KUKA KRL program: ps_p13060r5_ltc_geo_c1.src, ps_p13060r5_ltc_geo_c1.dat

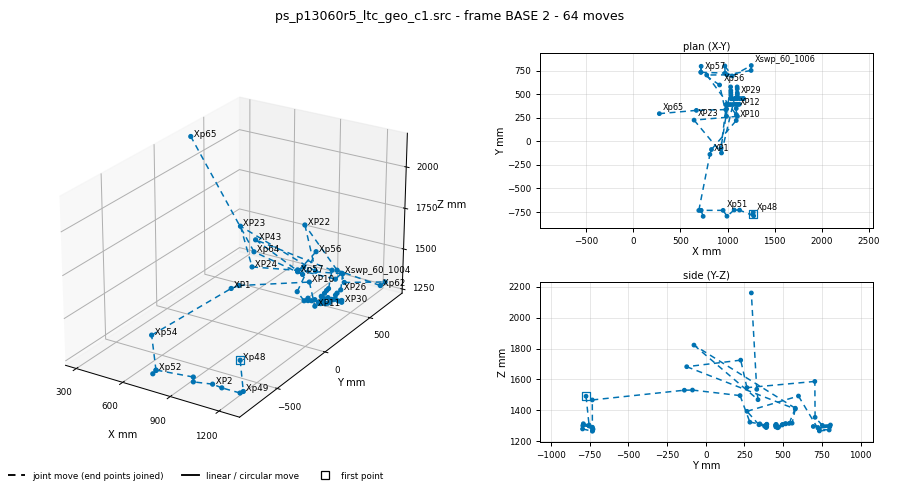
[picture p0: tool path of ps_p13060r5_ltc_geo_c1.src in frame BASE 2, 64 of 72 moves have a stored position in this frame; points joined in program order, loops and branches not executed]
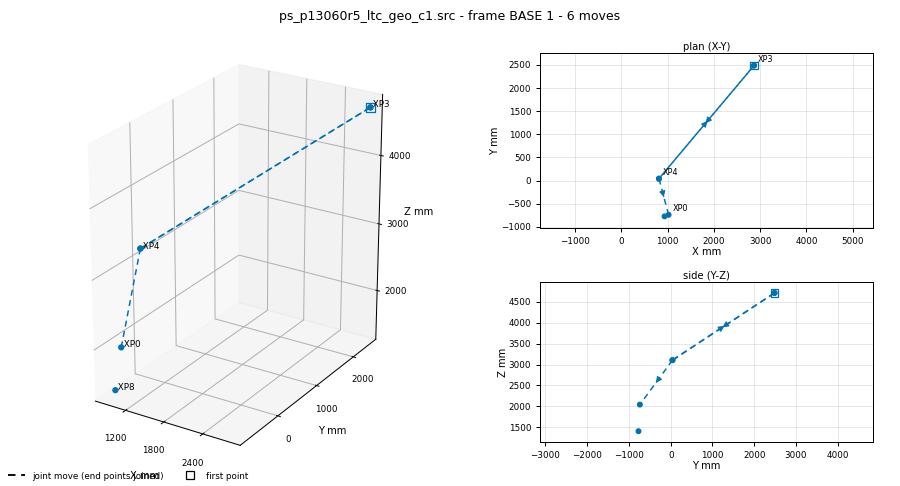
[picture p1: tool path of ps_p13060r5_ltc_geo_c1.src in frame BASE 1, 6 of 72 moves have a stored position in this frame; points joined in program order, loops and branches not executed]
--- ps_p13060r5_ltc_geo_c1.src ---
&ACCESS RVO2
&REL 201
&COMMENT SOLDA LTC  GUN C1
&PARAM DISKPATH = KRC:\R1\Program
DEF ps_p13060r5_ltc_geo_c1( )
;FOLD INI
  ;FOLD BASISTECH INI
    GLOBAL INTERRUPT DECL 3 WHEN $STOPMESS==TRUE DO IR_STOPM ( )
    INTERRUPT ON 3
    BAS (#INITMOV,0 )
  ;ENDFOLD (BASISTECH INI)
;FOLD SPOTTECH INI
USERSPOT(#INIT)
;ENDFOLD (SPOTTECH INI)
;FOLD GRIPPERTECH INI

;ENDFOLD (GRIPPERTECH INI)
  ;FOLD USER INI
    ;Make your modifications here

     ;FOLD COLLISION_V_3.01 INI ;%{E}
        IF (COLLISION_DATA[1].I_NR>0) THEN
          GLOBAL INTERRUPT DECL 21 WHEN $IN[COLLISION_DATA[1].I_NR]==FALSE DO COLLSTOP (1,0 )
        ENDIF
        IF (COLLISION_DATA[2].I_NR>0) THEN
          GLOBAL INTERRUPT DECL 22 WHEN $IN[COLLISION_DATA[2].I_NR]==FALSE DO COLLSTOP (2,0 )
        ENDIF
        IF (COLLISION_DATA[3].I_NR>0) THEN
          GLOBAL INTERRUPT DECL 23 WHEN $IN[COLLISION_DATA[3].I_NR]==FALSE DO COLLSTOP (3,0 )
        ENDIF
        IF (COLLISION_DATA[4].I_NR>0) THEN
          GLOBAL INTERRUPT DECL 24 WHEN $IN[COLLISION_DATA[4].I_NR]==FALSE DO COLLSTOP (4,0 )
        ENDIF
     ;ENDFOLD (Collision)

  ;ENDFOLD (USER INI)
;ENDFOLD (INI)

; Caracterização dos meios de produção: P13.060-R5
; Versão atual: 17/07/2013 Nome: Solda Geometria Accelo
; Change: C1

chk_w2_wechs_ok ( )           ; VERIFICAÇÃO DE FERRAMENA: C1

;FOLD PTP HOME Vel=100 % DEFAULT;%{PE}%R 8.2.20,%MKUKATPBASIS,%CMOVE,%VPTP,%P 1:PTP, 2:HOME, 3:, 5:100, 7:DEFAULT
$BWDSTART=FALSE
PDAT_ACT=PDEFAULT
FDAT_ACT=FHOME
BAS(#PTP_PARAMS,100)
$H_POS=XHOME
PTP XHOME
;ENDFOLD

IF(NOT(GHOST())) THEN

IF MaxStandMenge (1) THEN
 MaxStandmengeErreicht (1)
ENDIF

IF Elektrodenwechsel (1) THEN
 e_Fraes_2 ()   ; Fresa C1
ENDIF

ENDIF

;FOLD PTP P3 CONT Vel=75 % PDAT3 Tool[2]:Gun C1 Base[1]:Actros;%{PE}%R 8.2.20,%MKUKATPBASIS,%CMOVE,%VPTP,%P 1:PTP, 2:P3, 3:C_DIS, 5:75, 7:PDAT3
$BWDSTART=FALSE
PDAT_ACT=PPDAT3
FDAT_ACT=FP3
BAS(#PTP_PARAMS,75)
PTP XP3 C_DIS
;ENDFOLD
;FOLD PTP P4 CONT Vel=75 % PDAT4 Tool[2]:Gun C1 Base[1]:Actros;%{PE}%R 8.2.20,%MKUKATPBASIS,%CMOVE,%VPTP,%P 1:PTP, 2:P4, 3:C_DIS, 5:75, 7:PDAT4
$BWDSTART=FALSE
PDAT_ACT=PPDAT4
FDAT_ACT=FP4
BAS(#PTP_PARAMS,75)
PTP XP4 C_DIS
;ENDFOLD
;FOLD PTP P0 Vel=75 % PDAT0 Tool[2]:Gun C1 Base[1]:Actros;%{PE}%R 8.2.20,%MKUKATPBASIS,%CMOVE,%VPTP,%P 1:PTP, 2:P0, 3:, 5:75, 7:PDAT0
$BWDSTART=FALSE
PDAT_ACT=PPDAT0
FDAT_ACT=FP0
BAS(#PTP_PARAMS,75)
PTP XP0
;ENDFOLD

;FOLD OUT 3335 'R5 Solicit lib Soldar Geometria' State=TRUE ;%{PE}%R 8.2.20,%MKUKATPBASIS,%COUT,%VOUTX,%P 2:3335, 3:R5 Solicit lib Soldar Geometria, 5:TRUE, 6:
$OUT[3335]=TRUE
;ENDFOLD
;FOLD WAIT FOR ( IN 3339 'R5 GUARDA LIB. SOLDAR GEOMETRIA' );%{PE}%R 8.2.20,%MKUKATPBASIS,%CEXT_WAIT_FOR,%VEXT_WAIT_FOR,%P 2:, 4:, 5:$IN, 6:3339, 7:R5 GUARDA LIB. SOLDAR GEOMETRIA, 9:
WAIT FOR  ( $IN[3339] )
;ENDFOLD
;FOLD OUT 3335 'R5 Solicit lib Soldar Geometria' State=FALSE ;%{PE}%R 8.2.20,%MKUKATPBASIS,%COUT,%VOUTX,%P 2:3335, 3:R5 Solicit lib Soldar Geometria, 5:FALSE, 6:
$OUT[3335]=FALSE
;ENDFOLD

;FOLD PTP p48 CONT Vel=75 % P_OLP2 Tool[2]:Gun C1 Base[1]:Actros;%{PE}%R 8.2.20,%MKUKATPBASIS,%CMOVE,%VPTP,%P 1:PTP, 2:p48, 3:C_DIS, 5:75, 7:P_OLP2
$BWDSTART=FALSE
PDAT_ACT=PP_OLP2
FDAT_ACT=Fp48
BAS(#PTP_PARAMS,75)
PTP Xp48 C_DIS
;ENDFOLD

;FOLD OUT 3339 'R5 SOLDANDO' State=TRUE ;%{PE}%R 8.2.20,%MKUKATPBASIS,%COUT,%VOUTX,%P 2:3339, 3:R5 SOLDANDO, 5:TRUE, 6:
$OUT[3339]=TRUE
;ENDFOLD
;FOLD OUT 3340 'locking-signal PLC' State=FALSE ;%{PE}%R 8.2.20,%MKUKATPBASIS,%COUT,%VOUTX,%P 2:3340, 3:locking-signal PLC, 5:FALSE, 6:
$OUT[3340]=FALSE
;ENDFOLD

;FOLD PTP p49 CONT Vel=60 % P_OLP3 Tool[2]:Gun C1 Base[1]:Actros;%{PE}%R 8.2.20,%MKUKATPBASIS,%CMOVE,%VPTP,%P 1:PTP, 2:p49, 3:C_DIS, 5:60, 7:P_OLP3
$BWDSTART=FALSE
PDAT_ACT=PP_OLP3
FDAT_ACT=Fp49
BAS(#PTP_PARAMS,60)
PTP Xp49 C_DIS
;ENDFOLD

;FOLD ; SWP_60_1005;%{PE}%R8.2,%MKUKATPBASIS,%CCOMMENT,%VNORMAL,%P 2: SWP_60_1005
;ENDFOLD
;FOLD PTP swp_60_1005 P_OLP4 SPOT Gun=1 RETR OPN PgNo1=1 ACTIVE=1 Tool[2]:Gun C1 Base[2]:Accelo;%{PE}%R 8.2.2,%MKUKATPSPOT,%CSPOT,%VPTP,%P 1:PTP, 2:swp_60_1005, 3:, 5:100, 7:P_OLP4, 10:1, 12:#FIRST, 14:#OPN, 16:1, 18:1, 20:1, 22:0, 24:1, 25:S_OLP1
$BWDSTART=FALSE
PDAT_ACT=PP_OLP4
FDAT_ACT=Fswp_60_1005
BAS(#PTP_PARAMS,PP_OLP4.VEL)
S_ACT.GUN=1
S_ACT.PAIR=SDEFAULT.PAIR
S_ACT.RETR=#OPN
S_ACT.CLO_TM=1
S_ACT.PGNO1=1
S_ACT.PGNO2=SDEFAULT.PGNO2
S_ACT.PRESS1=SDEFAULT.PRESS1
S_ACT.PRESS2=SDEFAULT.PRESS2
S_READY=FALSE
PTP Xswp_60_1005
USERSPOT(#SPOT, S_ACT)
WAIT FOR S_READY
;ENDFOLD

;FOLD PTP p50 CONT Vel=60 % P_OLP5 Tool[2]:Gun C1 Base[1]:Actros;%{PE}%R 8.2.20,%MKUKATPBASIS,%CMOVE,%VPTP,%P 1:PTP, 2:p50, 3:C_DIS, 5:60, 7:P_OLP5
$BWDSTART=FALSE
PDAT_ACT=PP_OLP5
FDAT_ACT=Fp50
BAS(#PTP_PARAMS,60)
PTP Xp50 C_DIS
;ENDFOLD
;FOLD PTP P2 CONT Vel=60 % PDAT2 Tool[2]:Gun C1 Base[1]:Actros;%{PE}%R 8.2.20,%MKUKATPBASIS,%CMOVE,%VPTP,%P 1:PTP, 2:P2, 3:C_DIS, 5:60, 7:PDAT2
$BWDSTART=FALSE
PDAT_ACT=PPDAT2
FDAT_ACT=FP2
BAS(#PTP_PARAMS,60)
PTP XP2 C_DIS
;ENDFOLD

;FOLD ; SWP_60_1003;%{PE}%R8.2,%MKUKATPBASIS,%CCOMMENT,%VNORMAL,%P 2: SWP_60_1003
;ENDFOLD
;FOLD PTP swp_60_1003 P_OLP6 SPOT Gun=1 RETR OPN PgNo1=2 ACTIVE=1 Tool[2]:Gun C1 Base[2]:Accelo;%{PE}%R 8.2.2,%MKUKATPSPOT,%CSPOT,%VPTP,%P 1:PTP, 2:swp_60_1003, 3:, 5:100, 7:P_OLP6, 10:1, 12:#FIRST, 14:#OPN, 16:2, 18:1, 20:1, 22:0, 24:1, 25:S_OLP2
$BWDSTART=FALSE
PDAT_ACT=PP_OLP6
FDAT_ACT=Fswp_60_1003
BAS(#PTP_PARAMS,PP_OLP6.VEL)
S_ACT.GUN=1
S_ACT.PAIR=SDEFAULT.PAIR
S_ACT.RETR=#OPN
S_ACT.CLO_TM=1
S_ACT.PGNO1=2
S_ACT.PGNO2=SDEFAULT.PGNO2
S_ACT.PRESS1=SDEFAULT.PRESS1
S_ACT.PRESS2=SDEFAULT.PRESS2
S_READY=FALSE
PTP Xswp_60_1003
USERSPOT(#SPOT, S_ACT)
WAIT FOR S_READY
;ENDFOLD

;FOLD PTP p51 CONT Vel=60 % P_OLP7 Tool[2]:Gun C1 Base[1]:Actros;%{PE}%R 8.2.20,%MKUKATPBASIS,%CMOVE,%VPTP,%P 1:PTP, 2:p51, 3:C_DIS, 5:60, 7:P_OLP7
$BWDSTART=FALSE
PDAT_ACT=PP_OLP7
FDAT_ACT=Fp51
BAS(#PTP_PARAMS,60)
PTP Xp51 C_DIS
;ENDFOLD
;FOLD PTP p52 CONT Vel=60 % P_OLP8 Tool[2]:Gun C1 Base[1]:Actros;%{PE}%R 8.2.20,%MKUKATPBASIS,%CMOVE,%VPTP,%P 1:PTP, 2:p52, 3:C_DIS, 5:60, 7:P_OLP8
$BWDSTART=FALSE
PDAT_ACT=PP_OLP8
FDAT_ACT=Fp52
BAS(#PTP_PARAMS,60)
PTP Xp52 C_DIS
;ENDFOLD
;FOLD PTP P8 CONT Vel=100 % PDAT8 Tool[2]:Gun C1 Base[1]:Actros;%{PE}%R 8.2.20,%MKUKATPBASIS,%CMOVE,%VPTP,%P 1:PTP, 2:P8, 3:C_DIS, 5:100, 7:PDAT8
$BWDSTART=FALSE
PDAT_ACT=PPDAT8
FDAT_ACT=FP8
BAS(#PTP_PARAMS,100)
PTP XP8 C_DIS
;ENDFOLD

;FOLD ; SWP_60_1001;%{PE}%R8.2,%MKUKATPBASIS,%CCOMMENT,%VNORMAL,%P 2: SWP_60_1001
;ENDFOLD
;FOLD PTP swp_60_1001 P_OLP9 SPOT Gun=1 RETR OPN PgNo1=3 ACTIVE=1 Tool[2]:Gun C1 Base[2]:Accelo;%{PE}%R 8.2.2,%MKUKATPSPOT,%CSPOT,%VPTP,%P 1:PTP, 2:swp_60_1001, 3:, 5:100, 7:P_OLP9, 10:1, 12:#FIRST, 14:#OPN, 16:3, 18:1, 20:1, 22:0, 24:1, 25:S_OLP3
$BWDSTART=FALSE
PDAT_ACT=PP_OLP9
FDAT_ACT=Fswp_60_1001
BAS(#PTP_PARAMS,PP_OLP9.VEL)
S_ACT.GUN=1
S_ACT.PAIR=SDEFAULT.PAIR
S_ACT.RETR=#OPN
S_ACT.CLO_TM=1
S_ACT.PGNO1=3
S_ACT.PGNO2=SDEFAULT.PGNO2
S_ACT.PRESS1=SDEFAULT.PRESS1
S_ACT.PRESS2=SDEFAULT.PRESS2
S_READY=FALSE
PTP Xswp_60_1001
USERSPOT(#SPOT, S_ACT)
WAIT FOR S_READY
;ENDFOLD

;FOLD PTP p53 CONT Vel=60 % P_OLP10 Tool[2]:Gun C1 Base[1]:Actros;%{PE}%R 8.2.20,%MKUKATPBASIS,%CMOVE,%VPTP,%P 1:PTP, 2:p53, 3:C_DIS, 5:60, 7:P_OLP10
$BWDSTART=FALSE
PDAT_ACT=PP_OLP10
FDAT_ACT=Fp53
BAS(#PTP_PARAMS,60)
PTP Xp53 C_DIS
;ENDFOLD
;FOLD PTP p54 CONT Vel=80 % P_OLP11 Tool[2]:Gun C1 Base[1]:Actros;%{PE}%R 8.2.20,%MKUKATPBASIS,%CMOVE,%VPTP,%P 1:PTP, 2:p54, 3:C_DIS, 5:80, 7:P_OLP11
$BWDSTART=FALSE
PDAT_ACT=PP_OLP11
FDAT_ACT=Fp54
BAS(#PTP_PARAMS,80)
PTP Xp54 C_DIS
;ENDFOLD

;FOLD Collision.Monitoring_4_On ;%{PE}%MKUKATPUSER
COLLSTOP( 4, 1 ) ;Interrupt-Controlled
;ENDFOLD

;FOLD PTP P1 CONT Vel=80 % PDAT1 Tool[2]:Gun C1 Base[1]:Actros;%{PE}%R 8.2.20,%MKUKATPBASIS,%CMOVE,%VPTP,%P 1:PTP, 2:P1, 3:C_DIS, 5:80, 7:PDAT1
$BWDSTART=FALSE
PDAT_ACT=PPDAT1
FDAT_ACT=FP1
BAS(#PTP_PARAMS,80)
PTP XP1 C_DIS
;ENDFOLD
;FOLD PTP p55 CONT Vel=80 % P_OLP12 Tool[2]:Gun C1 Base[1]:Actros;%{PE}%R 8.2.20,%MKUKATPBASIS,%CMOVE,%VPTP,%P 1:PTP, 2:p55, 3:C_DIS, 5:80, 7:P_OLP12
$BWDSTART=FALSE
PDAT_ACT=PP_OLP12
FDAT_ACT=Fp55
BAS(#PTP_PARAMS,80)
PTP Xp55 C_DIS
;ENDFOLD
;FOLD PTP P10 CONT Vel=70 % PDAT10 Tool[2]:Gun C1 Base[1]:Actros;%{PE}%R 8.2.20,%MKUKATPBASIS,%CMOVE,%VPTP,%P 1:PTP, 2:P10, 3:C_DIS, 5:70, 7:PDAT10
$BWDSTART=FALSE
PDAT_ACT=PPDAT10
FDAT_ACT=FP10
BAS(#PTP_PARAMS,70)
PTP XP10 C_DIS
;ENDFOLD
;FOLD PTP P11 CONT Vel=70 % PDAT11 Tool[2]:Gun C1 Base[1]:Actros;%{PE}%R 8.2.20,%MKUKATPBASIS,%CMOVE,%VPTP,%P 1:PTP, 2:P11, 3:C_DIS, 5:70, 7:PDAT11
$BWDSTART=FALSE
PDAT_ACT=PPDAT11
FDAT_ACT=FP11
BAS(#PTP_PARAMS,70)
PTP XP11 C_DIS
;ENDFOLD
;FOLD PTP P12 CONT Vel=50 % PDAT12 Tool[2]:Gun C1 Base[1]:Actros;%{PE}%R 8.2.20,%MKUKATPBASIS,%CMOVE,%VPTP,%P 1:PTP, 2:P12, 3:C_DIS, 5:50, 7:PDAT12
$BWDSTART=FALSE
PDAT_ACT=PPDAT12
FDAT_ACT=FP12
BAS(#PTP_PARAMS,50)
PTP XP12 C_DIS
;ENDFOLD
;FOLD PTP P13 CONT Vel=50 % PDAT13 Tool[2]:Gun C1 Base[1]:Actros;%{PE}%R 8.2.20,%MKUKATPBASIS,%CMOVE,%VPTP,%P 1:PTP, 2:P13, 3:C_DIS, 5:50, 7:PDAT13
$BWDSTART=FALSE
PDAT_ACT=PPDAT13
FDAT_ACT=FP13
BAS(#PTP_PARAMS,50)
PTP XP13 C_DIS
;ENDFOLD


;FOLD PTP Swp_65_0004 PDAT14 SPOT Gun=1 RETR OPN PgNo1=7 ACTIVE=1 Tool[2]:Gun C1 Base[2]:Accelo;%{PE}%R 8.2.2,%MKUKATPSPOT,%CSPOT,%VPTP,%P 1:PTP, 2:Swp_65_0004, 3:, 5:70, 7:PDAT14, 10:1, 12:#FIRST, 14:#OPN, 16:7, 18:1, 20:0, 22:0, 24:1, 25:NORMAL
$BWDSTART=FALSE
PDAT_ACT=PPDAT14
FDAT_ACT=FSwp_65_0004
BAS(#PTP_PARAMS,PPDAT14.VEL)
S_ACT.GUN=1
S_ACT.PAIR=SDEFAULT.PAIR
S_ACT.RETR=#OPN
S_ACT.CLO_TM=1
S_ACT.PGNO1=7
S_ACT.PGNO2=SDEFAULT.PGNO2
S_ACT.PRESS1=SDEFAULT.PRESS1
S_ACT.PRESS2=SDEFAULT.PRESS2
S_READY=FALSE
PTP XSwp_65_0004
USERSPOT(#SPOT, S_ACT)
WAIT FOR S_READY
;ENDFOLD


;FOLD PTP P45 CONT Vel=50 % PDAT45 Tool[2]:Gun C1 Base[1]:Actros;%{PE}%R 8.2.20,%MKUKATPBASIS,%CMOVE,%VPTP,%P 1:PTP, 2:P45, 3:C_DIS, 5:50, 7:PDAT45
$BWDSTART=FALSE
PDAT_ACT=PPDAT45
FDAT_ACT=FP45
BAS(#PTP_PARAMS,50)
PTP XP45 C_DIS
;ENDFOLD


;FOLD PTP Swp_65_0006 PDAT15 SPOT Gun=1 RETR OPN PgNo1=8 ACTIVE=1 Tool[2]:Gun C1 Base[2]:Accelo;%{PE}%R 8.2.2,%MKUKATPSPOT,%CSPOT,%VPTP,%P 1:PTP, 2:Swp_65_0006, 3:, 5:70, 7:PDAT15, 10:1, 12:#FIRST, 14:#OPN, 16:8, 18:1, 20:0, 22:0, 24:1, 25:NORMAL
$BWDSTART=FALSE
PDAT_ACT=PPDAT15
FDAT_ACT=FSwp_65_0006
BAS(#PTP_PARAMS,PPDAT15.VEL)
S_ACT.GUN=1
S_ACT.PAIR=SDEFAULT.PAIR
S_ACT.RETR=#OPN
S_ACT.CLO_TM=1
S_ACT.PGNO1=8
S_ACT.PGNO2=SDEFAULT.PGNO2
S_ACT.PRESS1=SDEFAULT.PRESS1
S_ACT.PRESS2=SDEFAULT.PRESS2
S_READY=FALSE
PTP XSwp_65_0006
USERSPOT(#SPOT, S_ACT)
WAIT FOR S_READY
;ENDFOLD


;FOLD PTP P46 CONT Vel=50 % PDAT46 Tool[2]:Gun C1 Base[1]:Actros;%{PE}%R 8.2.20,%MKUKATPBASIS,%CMOVE,%VPTP,%P 1:PTP, 2:P46, 3:C_DIS, 5:50, 7:PDAT46
$BWDSTART=FALSE
PDAT_ACT=PPDAT46
FDAT_ACT=FP46
BAS(#PTP_PARAMS,50)
PTP XP46 C_DIS
;ENDFOLD


;FOLD PTP Swp_65_0008 PDAT16 SPOT Gun=1 RETR OPN PgNo1=9 ACTIVE=1 Tool[2]:Gun C1 Base[2]:Accelo;%{PE}%R 8.2.2,%MKUKATPSPOT,%CSPOT,%VPTP,%P 1:PTP, 2:Swp_65_0008, 3:, 5:70, 7:PDAT16, 10:1, 12:#FIRST, 14:#OPN, 16:9, 18:1, 20:0, 22:0, 24:1, 25:NORMAL
$BWDSTART=FALSE
PDAT_ACT=PPDAT16
FDAT_ACT=FSwp_65_0008
BAS(#PTP_PARAMS,PPDAT16.VEL)
S_ACT.GUN=1
S_ACT.PAIR=SDEFAULT.PAIR
S_ACT.RETR=#OPN
S_ACT.CLO_TM=1
S_ACT.PGNO1=9
S_ACT.PGNO2=SDEFAULT.PGNO2
S_ACT.PRESS1=SDEFAULT.PRESS1
S_ACT.PRESS2=SDEFAULT.PRESS2
S_READY=FALSE
PTP XSwp_65_0008
USERSPOT(#SPOT, S_ACT)
WAIT FOR S_READY
;ENDFOLD


;FOLD PTP P66 CONT Vel=50 % PDAT47 Tool[2]:Gun C1 Base[1]:Actros;%{PE}%R 8.2.20,%MKUKATPBASIS,%CMOVE,%VPTP,%P 1:PTP, 2:P66, 3:C_DIS, 5:50, 7:PDAT47
$BWDSTART=FALSE
PDAT_ACT=PPDAT47
FDAT_ACT=FP66
BAS(#PTP_PARAMS,50)
PTP XP66 C_DIS
;ENDFOLD


;FOLD PTP Swp_65_0010 PDAT17 SPOT Gun=1 RETR OPN PgNo1=10 ACTIVE=1 Tool[2]:Gun C1 Base[2]:Accelo;%{PE}%R 8.2.2,%MKUKATPSPOT,%CSPOT,%VPTP,%P 1:PTP, 2:Swp_65_0010, 3:, 5:70, 7:PDAT17, 10:1, 12:#FIRST, 14:#OPN, 16:10, 18:1, 20:0, 22:0, 24:1, 25:NORMAL
$BWDSTART=FALSE
PDAT_ACT=PPDAT17
FDAT_ACT=FSwp_65_0010
BAS(#PTP_PARAMS,PPDAT17.VEL)
S_ACT.GUN=1
S_ACT.PAIR=SDEFAULT.PAIR
S_ACT.RETR=#OPN
S_ACT.CLO_TM=1
S_ACT.PGNO1=10
S_ACT.PGNO2=SDEFAULT.PGNO2
S_ACT.PRESS1=SDEFAULT.PRESS1
S_ACT.PRESS2=SDEFAULT.PRESS2
S_READY=FALSE
PTP XSwp_65_0010
USERSPOT(#SPOT, S_ACT)
WAIT FOR S_READY
;ENDFOLD


;FOLD PTP P18 CONT Vel=50 % PDAT18 Tool[2]:Gun C1 Base[1]:Actros;%{PE}%R 8.2.20,%MKUKATPBASIS,%CMOVE,%VPTP,%P 1:PTP, 2:P18, 3:C_DIS, 5:50, 7:PDAT18
$BWDSTART=FALSE
PDAT_ACT=PPDAT18
FDAT_ACT=FP18
BAS(#PTP_PARAMS,50)
PTP XP18 C_DIS
;ENDFOLD
;FOLD PTP P19 CONT Vel=50 % PDAT19 Tool[2]:Gun C1 Base[1]:Actros;%{PE}%R 8.2.20,%MKUKATPBASIS,%CMOVE,%VPTP,%P 1:PTP, 2:P19, 3:C_DIS, 5:50, 7:PDAT19
$BWDSTART=FALSE
PDAT_ACT=PPDAT19
FDAT_ACT=FP19
BAS(#PTP_PARAMS,50)
PTP XP19 C_DIS
;ENDFOLD
;FOLD PTP P20 CONT Vel=50 % PDAT20 Tool[2]:Gun C1 Base[1]:Actros;%{PE}%R 8.2.20,%MKUKATPBASIS,%CMOVE,%VPTP,%P 1:PTP, 2:P20, 3:C_DIS, 5:50, 7:PDAT20
$BWDSTART=FALSE
PDAT_ACT=PPDAT20
FDAT_ACT=FP20
BAS(#PTP_PARAMS,50)
PTP XP20 C_DIS
;ENDFOLD
;FOLD PTP P21 CONT Vel=70 % PDAT21 Tool[2]:Gun C1 Base[1]:Actros;%{PE}%R 8.2.20,%MKUKATPBASIS,%CMOVE,%VPTP,%P 1:PTP, 2:P21, 3:C_DIS, 5:70, 7:PDAT21
$BWDSTART=FALSE
PDAT_ACT=PPDAT21
FDAT_ACT=FP21
BAS(#PTP_PARAMS,70)
PTP XP21 C_DIS
;ENDFOLD
;FOLD PTP p56 CONT Vel=80 % P_OLP13 Tool[2]:Gun C1 Base[1]:Actros;%{PE}%R 8.2.20,%MKUKATPBASIS,%CMOVE,%VPTP,%P 1:PTP, 2:p56, 3:C_DIS, 5:80, 7:P_OLP13
$BWDSTART=FALSE
PDAT_ACT=PP_OLP13
FDAT_ACT=Fp56
BAS(#PTP_PARAMS,80)
PTP Xp56 C_DIS
;ENDFOLD
;FOLD PTP p57 CONT Vel=80 % P_OLP14 Tool[2]:Gun C1 Base[1]:Actros;%{PE}%R 8.2.20,%MKUKATPBASIS,%CMOVE,%VPTP,%P 1:PTP, 2:p57, 3:C_DIS, 5:80, 7:P_OLP14
$BWDSTART=FALSE
PDAT_ACT=PP_OLP14
FDAT_ACT=Fp57
BAS(#PTP_PARAMS,80)
PTP Xp57 C_DIS
;ENDFOLD

;FOLD ; SWP_60_1002;%{PE}%R8.2,%MKUKATPBASIS,%CCOMMENT,%VNORMAL,%P 2: SWP_60_1002
;ENDFOLD
;FOLD PTP swp_60_1002 P_OLP15 SPOT Gun=1 RETR OPN PgNo1=4 ACTIVE=1 Tool[2]:Gun C1 Base[2]:Accelo;%{PE}%R 8.2.2,%MKUKATPSPOT,%CSPOT,%VPTP,%P 1:PTP, 2:swp_60_1002, 3:, 5:100, 7:P_OLP15, 10:1, 12:#FIRST, 14:#OPN, 16:4, 18:1, 20:1, 22:0, 24:1, 25:S_OLP4
$BWDSTART=FALSE
PDAT_ACT=PP_OLP15
FDAT_ACT=Fswp_60_1002
BAS(#PTP_PARAMS,PP_OLP15.VEL)
S_ACT.GUN=1
S_ACT.PAIR=SDEFAULT.PAIR
S_ACT.RETR=#OPN
S_ACT.CLO_TM=1
S_ACT.PGNO1=4
S_ACT.PGNO2=SDEFAULT.PGNO2
S_ACT.PRESS1=SDEFAULT.PRESS1
S_ACT.PRESS2=SDEFAULT.PRESS2
S_READY=FALSE
PTP Xswp_60_1002
USERSPOT(#SPOT, S_ACT)
WAIT FOR S_READY
;ENDFOLD

;FOLD PTP p58 CONT Vel=60 % P_OLP16 Tool[2]:Gun C1 Base[1]:Actros;%{PE}%R 8.2.20,%MKUKATPBASIS,%CMOVE,%VPTP,%P 1:PTP, 2:p58, 3:C_DIS, 5:60, 7:P_OLP16
$BWDSTART=FALSE
PDAT_ACT=PP_OLP16
FDAT_ACT=Fp58
BAS(#PTP_PARAMS,60)
PTP Xp58 C_DIS
;ENDFOLD
;FOLD PTP p59 CONT Vel=60 % P_OLP17 Tool[2]:Gun C1 Base[1]:Actros;%{PE}%R 8.2.20,%MKUKATPBASIS,%CMOVE,%VPTP,%P 1:PTP, 2:p59, 3:C_DIS, 5:60, 7:P_OLP17
$BWDSTART=FALSE
PDAT_ACT=PP_OLP17
FDAT_ACT=Fp59
BAS(#PTP_PARAMS,60)
PTP Xp59 C_DIS
;ENDFOLD

;FOLD ; SWP_60_1004;%{PE}%R8.2,%MKUKATPBASIS,%CCOMMENT,%VNORMAL,%P 2: SWP_60_1004
;ENDFOLD
;FOLD LIN swp_60_1004 CPDAT1 SPOT Gun=1 RETR OPN PgNo1=5 ACTIVE=1 Tool[2]:Gun C1 Base[2]:Accelo;%{PE}%R 8.2.2,%MKUKATPSPOT,%CSPOT,%VLIN,%P 1:LIN, 2:swp_60_1004, 3:, 5:2, 7:CPDAT1, 10:1, 12:#FIRST, 14:#OPN, 16:5, 18:1, 20:1, 22:0, 24:1, 25:S_OLP5
$BWDSTART=FALSE
LDAT_ACT=LCPDAT1
FDAT_ACT=Fswp_60_1004
BAS(#CP_PARAMS,LCPDAT1.VEL)
S_ACT.GUN=1
S_ACT.PAIR=SDEFAULT.PAIR
S_ACT.RETR=#OPN
S_ACT.CLO_TM=1
S_ACT.PGNO1=5
S_ACT.PGNO2=SDEFAULT.PGNO2
S_ACT.PRESS1=SDEFAULT.PRESS1
S_ACT.PRESS2=SDEFAULT.PRESS2
S_READY=FALSE
LIN Xswp_60_1004
USERSPOT(#SPOT, S_ACT)
WAIT FOR S_READY
;ENDFOLD

;FOLD Collision.Monitoring_4_Off . ;%{PE}%MKUKATPUSER
COLLSTOP( 4, 2+0 )
;ENDFOLD

;FOLD PTP p61 CONT Vel=60 % P_OLP20 Tool[2]:Gun C1 Base[1]:Actros;%{PE}%R 8.2.20,%MKUKATPBASIS,%CMOVE,%VPTP,%P 1:PTP, 2:p61, 3:C_DIS, 5:60, 7:P_OLP20
$BWDSTART=FALSE
PDAT_ACT=PP_OLP20
FDAT_ACT=Fp61
BAS(#PTP_PARAMS,60)
PTP Xp61 C_DIS
;ENDFOLD

;FOLD ; SWP_60_1006;%{PE}%R8.2,%MKUKATPBASIS,%CCOMMENT,%VNORMAL,%P 2: SWP_60_1006
;ENDFOLD
;FOLD PTP swp_60_1006 P_OLP21 SPOT Gun=1 RETR OPN PgNo1=6 ACTIVE=1 Tool[2]:Gun C1 Base[2]:Accelo;%{PE}%R 8.2.2,%MKUKATPSPOT,%CSPOT,%VPTP,%P 1:PTP, 2:swp_60_1006, 3:, 5:100, 7:P_OLP21, 10:1, 12:#FIRST, 14:#OPN, 16:6, 18:1, 20:1, 22:0, 24:1, 25:S_OLP6
$BWDSTART=FALSE
PDAT_ACT=PP_OLP21
FDAT_ACT=Fswp_60_1006
BAS(#PTP_PARAMS,PP_OLP21.VEL)
S_ACT.GUN=1
S_ACT.PAIR=SDEFAULT.PAIR
S_ACT.RETR=#OPN
S_ACT.CLO_TM=1
S_ACT.PGNO1=6
S_ACT.PGNO2=SDEFAULT.PGNO2
S_ACT.PRESS1=SDEFAULT.PRESS1
S_ACT.PRESS2=SDEFAULT.PRESS2
S_READY=FALSE
PTP Xswp_60_1006
USERSPOT(#SPOT, S_ACT)
WAIT FOR S_READY
;ENDFOLD

;FOLD PTP p62 CONT Vel=60 % P_OLP22 Tool[2]:Gun C1 Base[1]:Actros;%{PE}%R 8.2.20,%MKUKATPBASIS,%CMOVE,%VPTP,%P 1:PTP, 2:p62, 3:C_DIS, 5:60, 7:P_OLP22
$BWDSTART=FALSE
PDAT_ACT=PP_OLP22
FDAT_ACT=Fp62
BAS(#PTP_PARAMS,60)
PTP Xp62 C_DIS
;ENDFOLD
;FOLD PTP p63 CONT Vel=60 % P_OLP23 Tool[2]:Gun C1 Base[1]:Actros;%{PE}%R 8.2.20,%MKUKATPBASIS,%CMOVE,%VPTP,%P 1:PTP, 2:p63, 3:C_DIS, 5:60, 7:P_OLP23
$BWDSTART=FALSE
PDAT_ACT=PP_OLP23
FDAT_ACT=Fp63
BAS(#PTP_PARAMS,60)
PTP Xp63 C_DIS
;ENDFOLD
;FOLD PTP P22 CONT Vel=70 % PDAT22 Tool[2]:Gun C1 Base[1]:Actros;%{PE}%R 8.2.20,%MKUKATPBASIS,%CMOVE,%VPTP,%P 1:PTP, 2:P22, 3:C_DIS, 5:70, 7:PDAT22
$BWDSTART=FALSE
PDAT_ACT=PPDAT22
FDAT_ACT=FP22
BAS(#PTP_PARAMS,70)
PTP XP22 C_DIS
;ENDFOLD
;FOLD PTP P67 CONT Vel=50 % PDAT48 Tool[2]:Gun C1 Base[1]:Actros;%{PE}%R 8.2.20,%MKUKATPBASIS,%CMOVE,%VPTP,%P 1:PTP, 2:P67, 3:C_DIS, 5:50, 7:PDAT48
$BWDSTART=FALSE
PDAT_ACT=PPDAT48
FDAT_ACT=FP67
BAS(#PTP_PARAMS,50)
PTP XP67 C_DIS
;ENDFOLD
;FOLD PTP P23 CONT Vel=50 % PDAT23 Tool[2]:Gun C1 Base[1]:Actros;%{PE}%R 8.2.20,%MKUKATPBASIS,%CMOVE,%VPTP,%P 1:PTP, 2:P23, 3:C_DIS, 5:50, 7:PDAT23
$BWDSTART=FALSE
PDAT_ACT=PPDAT23
FDAT_ACT=FP23
BAS(#PTP_PARAMS,50)
PTP XP23 C_DIS
;ENDFOLD
;FOLD PTP P24 CONT Vel=70 % PDAT24 Tool[2]:Gun C1 Base[1]:Actros;%{PE}%R 8.2.20,%MKUKATPBASIS,%CMOVE,%VPTP,%P 1:PTP, 2:P24, 3:C_DIS, 5:70, 7:PDAT24
$BWDSTART=FALSE
PDAT_ACT=PPDAT24
FDAT_ACT=FP24
BAS(#PTP_PARAMS,70)
PTP XP24 C_DIS
;ENDFOLD
;FOLD PTP P25 CONT Vel=70 % PDAT25 Tool[2]:Gun C1 Base[1]:Actros;%{PE}%R 8.2.20,%MKUKATPBASIS,%CMOVE,%VPTP,%P 1:PTP, 2:P25, 3:C_DIS, 5:70, 7:PDAT25
$BWDSTART=FALSE
PDAT_ACT=PPDAT25
FDAT_ACT=FP25
BAS(#PTP_PARAMS,70)
PTP XP25 C_DIS
;ENDFOLD
;FOLD PTP P26 CONT Vel=50 % PDAT26 Tool[2]:Gun C1 Base[1]:Actros;%{PE}%R 8.2.20,%MKUKATPBASIS,%CMOVE,%VPTP,%P 1:PTP, 2:P26, 3:C_DIS, 5:50, 7:PDAT26
$BWDSTART=FALSE
PDAT_ACT=PPDAT26
FDAT_ACT=FP26
BAS(#PTP_PARAMS,50)
PTP XP26 C_DIS
;ENDFOLD
;FOLD PTP P27 CONT Vel=50 % PDAT27 Tool[2]:Gun C1 Base[1]:Actros;%{PE}%R 8.2.20,%MKUKATPBASIS,%CMOVE,%VPTP,%P 1:PTP, 2:P27, 3:C_DIS, 5:50, 7:PDAT27
$BWDSTART=FALSE
PDAT_ACT=PPDAT27
FDAT_ACT=FP27
BAS(#PTP_PARAMS,50)
PTP XP27 C_DIS
;ENDFOLD
;FOLD PTP P28 CONT Vel=50 % PDAT28 Tool[2]:Gun C1 Base[1]:Actros;%{PE}%R 8.2.20,%MKUKATPBASIS,%CMOVE,%VPTP,%P 1:PTP, 2:P28, 3:C_DIS, 5:50, 7:PDAT28
$BWDSTART=FALSE
PDAT_ACT=PPDAT28
FDAT_ACT=FP28
BAS(#PTP_PARAMS,50)
PTP XP28 C_DIS
;ENDFOLD
;FOLD PTP P29 CONT Vel=50 % PDAT29 Tool[2]:Gun C1 Base[1]:Actros;%{PE}%R 8.2.20,%MKUKATPBASIS,%CMOVE,%VPTP,%P 1:PTP, 2:P29, 3:C_DIS, 5:50, 7:PDAT29
$BWDSTART=FALSE
PDAT_ACT=PPDAT29
FDAT_ACT=FP29
BAS(#PTP_PARAMS,50)
PTP XP29 C_DIS
;ENDFOLD
;FOLD PTP P30 CONT Vel=50 % PDAT30 Tool[2]:Gun C1 Base[1]:Actros;%{PE}%R 8.2.20,%MKUKATPBASIS,%CMOVE,%VPTP,%P 1:PTP, 2:P30, 3:C_DIS, 5:50, 7:PDAT30
$BWDSTART=FALSE
PDAT_ACT=PPDAT30
FDAT_ACT=FP30
BAS(#PTP_PARAMS,50)
PTP XP30 C_DIS
;ENDFOLD


;FOLD PTP Swp_65_0001 PDAT31 SPOT Gun=1 RETR OPN PgNo1=11 ACTIVE=1 Tool[2]:Gun C1 Base[2]:Accelo;%{PE}%R 8.2.2,%MKUKATPSPOT,%CSPOT,%VPTP,%P 1:PTP, 2:Swp_65_0001, 3:, 5:50, 7:PDAT31, 10:1, 12:#FIRST, 14:#OPN, 16:11, 18:1, 20:0, 22:0, 24:1, 25:NORMAL
$BWDSTART=FALSE
PDAT_ACT=PPDAT31
FDAT_ACT=FSwp_65_0001
BAS(#PTP_PARAMS,PPDAT31.VEL)
S_ACT.GUN=1
S_ACT.PAIR=SDEFAULT.PAIR
S_ACT.RETR=#OPN
S_ACT.CLO_TM=1
S_ACT.PGNO1=11
S_ACT.PGNO2=SDEFAULT.PGNO2
S_ACT.PRESS1=SDEFAULT.PRESS1
S_ACT.PRESS2=SDEFAULT.PRESS2
S_READY=FALSE
PTP XSwp_65_0001
USERSPOT(#SPOT, S_ACT)
WAIT FOR S_READY
;ENDFOLD


;FOLD PTP P32 Vel=50 % PDAT32 Tool[2]:Gun C1 Base[2]:Accelo;%{PE}%R 8.2.20,%MKUKATPBASIS,%CMOVE,%VPTP,%P 1:PTP, 2:P32, 3:, 5:50, 7:PDAT32
$BWDSTART=FALSE
PDAT_ACT=PPDAT32
FDAT_ACT=FP32
BAS(#PTP_PARAMS,50)
PTP XP32
;ENDFOLD


;FOLD PTP Swp_65_0003 PDAT33 SPOT Gun=1 RETR OPN PgNo1=12 ACTIVE=1 Tool[2]:Gun C1 Base[2]:Accelo;%{PE}%R 8.2.2,%MKUKATPSPOT,%CSPOT,%VPTP,%P 1:PTP, 2:Swp_65_0003, 3:, 5:50, 7:PDAT33, 10:1, 12:#FIRST, 14:#OPN, 16:12, 18:1, 20:0, 22:0, 24:1, 25:NORMAL
$BWDSTART=FALSE
PDAT_ACT=PPDAT33
FDAT_ACT=FSwp_65_0003
BAS(#PTP_PARAMS,PPDAT33.VEL)
S_ACT.GUN=1
S_ACT.PAIR=SDEFAULT.PAIR
S_ACT.RETR=#OPN
S_ACT.CLO_TM=1
S_ACT.PGNO1=12
S_ACT.PGNO2=SDEFAULT.PGNO2
S_ACT.PRESS1=SDEFAULT.PRESS1
S_ACT.PRESS2=SDEFAULT.PRESS2
S_READY=FALSE
PTP XSwp_65_0003
USERSPOT(#SPOT, S_ACT)
WAIT FOR S_READY
;ENDFOLD


;FOLD PTP P34 Vel=50 % PDAT34 Tool[2]:Gun C1 Base[2]:Accelo;%{PE}%R 8.2.20,%MKUKATPBASIS,%CMOVE,%VPTP,%P 1:PTP, 2:P34, 3:, 5:50, 7:PDAT34
$BWDSTART=FALSE
PDAT_ACT=PPDAT34
FDAT_ACT=FP34
BAS(#PTP_PARAMS,50)
PTP XP34
;ENDFOLD


;FOLD PTP Swp_65_0005 PDAT35 SPOT Gun=1 RETR OPN PgNo1=13 ACTIVE=1 Tool[2]:Gun C1 Base[2]:Accelo;%{PE}%R 8.2.2,%MKUKATPSPOT,%CSPOT,%VPTP,%P 1:PTP, 2:Swp_65_0005, 3:, 5:50, 7:PDAT35, 10:1, 12:#FIRST, 14:#OPN, 16:13, 18:1, 20:0, 22:0, 24:1, 25:NORMAL
$BWDSTART=FALSE
PDAT_ACT=PPDAT35
FDAT_ACT=FSwp_65_0005
BAS(#PTP_PARAMS,PPDAT35.VEL)
S_ACT.GUN=1
S_ACT.PAIR=SDEFAULT.PAIR
S_ACT.RETR=#OPN
S_ACT.CLO_TM=1
S_ACT.PGNO1=13
S_ACT.PGNO2=SDEFAULT.PGNO2
S_ACT.PRESS1=SDEFAULT.PRESS1
S_ACT.PRESS2=SDEFAULT.PRESS2
S_READY=FALSE
PTP XSwp_65_0005
USERSPOT(#SPOT, S_ACT)
WAIT FOR S_READY
;ENDFOLD


;FOLD PTP P36 Vel=50 % PDAT36 Tool[2]:Gun C1 Base[2]:Accelo;%{PE}%R 8.2.20,%MKUKATPBASIS,%CMOVE,%VPTP,%P 1:PTP, 2:P36, 3:, 5:50, 7:PDAT36
$BWDSTART=FALSE
PDAT_ACT=PPDAT36
FDAT_ACT=FP36
BAS(#PTP_PARAMS,50)
PTP XP36
;ENDFOLD


;FOLD PTP Swp_65_0007 PDAT37 SPOT Gun=1 RETR OPN PgNo1=14 ACTIVE=1 Tool[2]:Gun C1 Base[2]:Accelo;%{PE}%R 8.2.2,%MKUKATPSPOT,%CSPOT,%VPTP,%P 1:PTP, 2:Swp_65_0007, 3:, 5:50, 7:PDAT37, 10:1, 12:#FIRST, 14:#OPN, 16:14, 18:1, 20:0, 22:0, 24:1, 25:NORMAL
$BWDSTART=FALSE
PDAT_ACT=PPDAT37
FDAT_ACT=FSwp_65_0007
BAS(#PTP_PARAMS,PPDAT37.VEL)
S_ACT.GUN=1
S_ACT.PAIR=SDEFAULT.PAIR
S_ACT.RETR=#OPN
S_ACT.CLO_TM=1
S_ACT.PGNO1=14
S_ACT.PGNO2=SDEFAULT.PGNO2
S_ACT.PRESS1=SDEFAULT.PRESS1
S_ACT.PRESS2=SDEFAULT.PRESS2
S_READY=FALSE
PTP XSwp_65_0007
USERSPOT(#SPOT, S_ACT)
WAIT FOR S_READY
;ENDFOLD


;FOLD PTP P38 Vel=50 % PDAT38 Tool[2]:Gun C1 Base[2]:Accelo;%{PE}%R 8.2.20,%MKUKATPBASIS,%CMOVE,%VPTP,%P 1:PTP, 2:P38, 3:, 5:50, 7:PDAT38
$BWDSTART=FALSE
PDAT_ACT=PPDAT38
FDAT_ACT=FP38
BAS(#PTP_PARAMS,50)
PTP XP38
;ENDFOLD
;FOLD PTP P39 Vel=50 % PDAT39 Tool[2]:Gun C1 Base[2]:Accelo;%{PE}%R 8.2.20,%MKUKATPBASIS,%CMOVE,%VPTP,%P 1:PTP, 2:P39, 3:, 5:50, 7:PDAT39
$BWDSTART=FALSE
PDAT_ACT=PPDAT39
FDAT_ACT=FP39
BAS(#PTP_PARAMS,50)
PTP XP39
;ENDFOLD
;FOLD PTP P40 Vel=50 % PDAT40 Tool[2]:Gun C1 Base[2]:Accelo;%{PE}%R 8.2.20,%MKUKATPBASIS,%CMOVE,%VPTP,%P 1:PTP, 2:P40, 3:, 5:50, 7:PDAT40
$BWDSTART=FALSE
PDAT_ACT=PPDAT40
FDAT_ACT=FP40
BAS(#PTP_PARAMS,50)
PTP XP40
;ENDFOLD
;FOLD PTP P41 Vel=50 % PDAT41 Tool[2]:Gun C1 Base[2]:Accelo;%{PE}%R 8.2.20,%MKUKATPBASIS,%CMOVE,%VPTP,%P 1:PTP, 2:P41, 3:, 5:50, 7:PDAT41
$BWDSTART=FALSE
PDAT_ACT=PPDAT41
FDAT_ACT=FP41
BAS(#PTP_PARAMS,50)
PTP XP41
;ENDFOLD
;FOLD PTP P42 Vel=50 % PDAT42 Tool[2]:Gun C1 Base[2]:Accelo;%{PE}%R 8.2.20,%MKUKATPBASIS,%CMOVE,%VPTP,%P 1:PTP, 2:P42, 3:, 5:50, 7:PDAT42
$BWDSTART=FALSE
PDAT_ACT=PPDAT42
FDAT_ACT=FP42
BAS(#PTP_PARAMS,50)
PTP XP42
;ENDFOLD
;FOLD PTP P43 CONT Vel=50 % PDAT43 Tool[2]:Gun C1 Base[1]:Actros;%{PE}%R 8.2.20,%MKUKATPBASIS,%CMOVE,%VPTP,%P 1:PTP, 2:P43, 3:C_DIS, 5:50, 7:PDAT43
$BWDSTART=FALSE
PDAT_ACT=PPDAT43
FDAT_ACT=FP43
BAS(#PTP_PARAMS,50)
PTP XP43 C_DIS
;ENDFOLD
;FOLD PTP P44 CONT Vel=50 % PDAT44 Tool[2]:Gun C1 Base[1]:Actros;%{PE}%R 8.2.20,%MKUKATPBASIS,%CMOVE,%VPTP,%P 1:PTP, 2:P44, 3:C_DIS, 5:50, 7:PDAT44
$BWDSTART=FALSE
PDAT_ACT=PPDAT44
FDAT_ACT=FP44
BAS(#PTP_PARAMS,50)
PTP XP44 C_DIS
;ENDFOLD

;FOLD OUT 3339 'R5 SOLDANDO' State=FALSE ;%{PE}%R 8.2.20,%MKUKATPBASIS,%COUT,%VOUTX,%P 2:3339, 3:R5 SOLDANDO, 5:FALSE, 6:
$OUT[3339]=FALSE
;ENDFOLD
;FOLD OUT 3340 'locking-signal PLC' State=TRUE ;%{PE}%R 8.2.20,%MKUKATPBASIS,%COUT,%VOUTX,%P 2:3340, 3:locking-signal PLC, 5:TRUE, 6:
$OUT[3340]=TRUE
;ENDFOLD

;FOLD PULSE 3338 'R5 SOLDA GEOMETRIA ACCELO OK' State=TRUE Time=3 sec;%{PE}%R 8.2.20,%MKUKATPBASIS,%COUT,%VPULSE,%P 2:3338, 3:R5 SOLDA GEOMETRIA ACCELO OK, 5:TRUE, 6:, 8:3
PULSE($OUT[3338], TRUE,3)
;ENDFOLD

;FOLD PTP p64 CONT Vel=70 % P_OLP24 Tool[2]:Gun C1 Base[1]:Actros;%{PE}%R 8.2.20,%MKUKATPBASIS,%CMOVE,%VPTP,%P 1:PTP, 2:p64, 3:C_DIS, 5:70, 7:P_OLP24
$BWDSTART=FALSE
PDAT_ACT=PP_OLP24
FDAT_ACT=Fp64
BAS(#PTP_PARAMS,70)
PTP Xp64 C_DIS
;ENDFOLD
;FOLD PTP p65 Vel=85 % P_OLP25 Tool[2]:Gun C1 Base[2]:Accelo;%{PE}%R 8.2.20,%MKUKATPBASIS,%CMOVE,%VPTP,%P 1:PTP, 2:p65, 3:, 5:85, 7:P_OLP25
$BWDSTART=FALSE
PDAT_ACT=PP_OLP25
FDAT_ACT=Fp65
BAS(#PTP_PARAMS,85)
PTP Xp65
;ENDFOLD
;FOLD PTP P5 CONT Vel=85 % PDAT5 Tool[2]:Gun C1 Base[1]:Actros;%{PE}%R 8.2.20,%MKUKATPBASIS,%CMOVE,%VPTP,%P 1:PTP, 2:P5, 3:C_DIS, 5:85, 7:PDAT5
$BWDSTART=FALSE
PDAT_ACT=PPDAT5
FDAT_ACT=FP5
BAS(#PTP_PARAMS,85)
PTP XP5 C_DIS
;ENDFOLD
;FOLD PTP P6 CONT Vel=85 % PDAT6 Tool[2]:Gun C1 Base[1]:Actros;%{PE}%R 8.2.20,%MKUKATPBASIS,%CMOVE,%VPTP,%P 1:PTP, 2:P6, 3:C_DIS, 5:85, 7:PDAT6
$BWDSTART=FALSE
PDAT_ACT=PPDAT6
FDAT_ACT=FP6
BAS(#PTP_PARAMS,85)
PTP XP6 C_DIS
;ENDFOLD

;FOLD PTP HOME Vel=85 % DEFAULT;%{PE}%R 8.2.20,%MKUKATPBASIS,%CMOVE,%VPTP,%P 1:PTP, 2:HOME, 3:, 5:85, 7:DEFAULT
$BWDSTART=FALSE
PDAT_ACT=PDEFAULT
FDAT_ACT=FHOME
BAS(#PTP_PARAMS,85)
$H_POS=XHOME
PTP XHOME
;ENDFOLD

IF (NOT(GHOST())) THEN

IF FraesAnf (1) THEN
 f_Fraes_2()   ; Fresa C1
ENDIF

ENDIF


END

--- ps_p13060r5_ltc_geo_c1.dat ---
&ACCESS RVO2
&REL 201
&COMMENT SOLDA LTC  GUN C1
&PARAM DISKPATH = KRC:\R1\Program
DEFDAT  ps_p13060r5_ltc_geo_c1
;FOLD EXTERNAL DECLARATIONS;%{PE}%MKUKATPBASIS,%CEXT,%VCOMMON,%P
;FOLD GRIPPERTECH EXT
EXT  H50 (INT  :IN,INT  :IN,INT  :IN,GRP_TYP  :IN )
;ENDFOLD (GRIPPERTECH EXT)
;FOLD SPOTTECH EXT
EXT  USERSPOT (S_COMMAND  :IN,SPOT_TYPE  :IN )
;ENDFOLD (SPOTTECH EXT)
;FOLD BASISTECH EXT;%{PE}%MKUKATPBASIS,%CEXT,%VEXT,%P
EXT  BAS (BAS_COMMAND  :IN,REAL  :IN )
DECL INT SUCCESS
;ENDFOLD (BASISTECH EXT)
;FOLD USER EXT;%{E}%MKUKATPUSER,%CEXT,%VEXT,%P
;Make your modifications here

;ENDFOLD (USER EXT)
;ENDFOLD (EXTERNAL DECLARATIONS)

;# ============ START PATH : swp_p13060r5_ltc_geo_c1 =============
DECL FDAT Fp48={TOOL_NO 2,BASE_NO 2,IPO_FRAME #BASE,POINT2[] " "}
DECL PDAT PP_OLP2={VEL 100.0,ACC 100.0,APO_DIST 100.0,APO_MODE #CDIS}
DECL E6POS Xp48={X 1267.16602,Y -773.572998,Z 1491.776,A -44.9560013,B 3.00539994,C 5.83080006,S 2,T 11}
DECL FDAT Fp49={TOOL_NO 2,BASE_NO 2,IPO_FRAME #BASE,POINT2[] " "}
DECL PDAT PP_OLP3={VEL 100.0,ACC 100.0,APO_DIST 100.0,APO_MODE #CDIS}
DECL E6POS Xp49={X 1273.53503,Y -753.973328,Z 1305.45496,A -44.9560013,B 3.00530005,C 5.83080006,S 2,T 11,E1 0.0,E2 0.0,E3 0.0,E4 0.0,E5 0.0,E6 0.0}
DECL FDAT Fswp_60_1005={TOOL_NO 2,BASE_NO 2,IPO_FRAME #BASE,POINT2[] " ",TQ_STATE FALSE}
DECL PDAT PP_OLP4={VEL 70.0,ACC 100.0,APO_DIST 0.0}
DECL SPOT_TYPE SS_OLP1={GUN 2,PAIR #FIRST,RETR #CLO,CLO_TM 0,PGNO1 1,PRESS1 1.0,PGNO2 0,PRESS2 0.0}
DECL E6POS Xswp_60_1005={X 1277.29895,Y -791.007507,Z 1314.19995,A -45.2053108,B 1.41634095,C 2.95584607,S 2,T 11,E1 0.0,E2 0.0,E3 0.0,E4 0.0,E5 0.0,E6 0.0}
DECL FDAT Fp50={TOOL_NO 2,BASE_NO 2,IPO_FRAME #BASE,POINT2[] " "}
DECL PDAT PP_OLP5={VEL 100.0,ACC 100.0,APO_DIST 100.0,APO_MODE #CDIS}
DECL E6POS Xp50={X 1127.45996,Y -729.703125,Z 1275.07605,A -45.0816803,B 0.418681502,C 2.49454689,S 2,T 11,E1 0.0,E2 0.0,E3 0.0,E4 0.0,E5 0.0,E6 0.0}
DECL FDAT Fswp_60_1003={TOOL_NO 2,BASE_NO 2,IPO_FRAME #BASE,POINT2[] " "}
DECL PDAT PP_OLP6={VEL 60.0,ACC 100.0,APO_DIST 0.0}
DECL SPOT_TYPE SS_OLP2={GUN 2,PAIR #FIRST,RETR #CLO,CLO_TM 0,PGNO1 1,PRESS1 1.0,PGNO2 0,PRESS2 0.0}
DECL E6POS Xswp_60_1003={X 993.994873,Y -794.501526,Z 1301.71899,A -76.0846329,B 3.40040302,C 4.36868286,S 2,T 11,E1 0.0,E2 0.0,E3 0.0,E4 0.0,E5 0.0,E6 0.0}
DECL FDAT Fp51={TOOL_NO 2,BASE_NO 2,IPO_FRAME #BASE,POINT2[] " "}
DECL PDAT PP_OLP7={VEL 100.0,ACC 100.0,APO_DIST 100.0,APO_MODE #CDIS}
DECL E6POS Xp51={X 953.202087,Y -732.422485,Z 1291.46204,A -75.9682999,B 4.97650003,C 4.5314002,S 2,T 11,E1 0.0,E2 0.0,E3 0.0,E4 0.0,E5 0.0,E6 0.0}
DECL FDAT Fp52={TOOL_NO 2,BASE_NO 2,IPO_FRAME #BASE,POINT2[] " "}
DECL PDAT PP_OLP8={VEL 100.0,ACC 100.0,APO_DIST 100.0,APO_MODE #CDIS}
DECL E6POS Xp52={X 718.411316,Y -732.486816,Z 1268.46204,A -89.3901062,B 5.38820982,C 6.46161318,S 2,T 11,E1 0.0,E2 0.0,E3 0.0,E4 0.0,E5 0.0,E6 0.0}
DECL FDAT Fswp_60_1001={TOOL_NO 2,BASE_NO 2,IPO_FRAME #BASE,POINT2[] " "}
DECL PDAT PP_OLP9={VEL 60.0,ACC 100.0,APO_DIST 0.0}
DECL SPOT_TYPE SS_OLP3={GUN 2,PAIR #FIRST,RETR #CLO,CLO_TM 0,PGNO1 1,PRESS1 1.0,PGNO2 0,PRESS2 0.0}
DECL E6POS Xswp_60_1001={X 741.385376,Y -796.038574,Z 1280.33606,A -102.193298,B 1.68797004,C 5.37691689,S 2,T 11,E1 0.0,E2 0.0,E3 0.0,E4 0.0,E5 0.0,E6 0.0}
DECL FDAT Fp53={TOOL_NO 2,BASE_NO 2,IPO_FRAME #BASE,POINT2[] " "}
DECL PDAT PP_OLP10={VEL 100.0,ACC 100.0,APO_DIST 100.0,APO_MODE #CDIS}
DECL E6POS Xp53={X 718.469421,Y -732.476013,Z 1265.88196,A -104.7658,B 6.90543222,C 4.8060112,S 2,T 11,E1 0.0,E2 0.0,E3 0.0,E4 0.0,E5 0.0,E6 0.0}
DECL FDAT Fp54={TOOL_NO 2,BASE_NO 2,IPO_FRAME #BASE,POINT2[] " "}
DECL PDAT PP_OLP11={VEL 100.0,ACC 100.0,APO_DIST 100.0,APO_MODE #CDIS}
DECL E6POS Xp54={X 695.093018,Y -733.262024,Z 1467.776,A -89.6514969,B 5.44920015,C 3.70050001,S 2,T 10}
DECL FDAT Fp55={TOOL_NO 2,BASE_NO 2,IPO_FRAME #BASE,POINT2[] " "}
DECL PDAT PP_OLP12={VEL 100.0,ACC 100.0,APO_DIST 100.0,APO_MODE #CDIS}
DECL E6POS Xp55={X 829.557983,Y -86.1466599,Z 1531.63306,A 104.081802,B 40.8783913,C 7.29571676,S 6,T 59,E1 0.0,E2 0.0,E3 0.0,E4 0.0,E5 0.0,E6 0.0}
DECL FDAT Fp56={TOOL_NO 2,BASE_NO 2,IPO_FRAME #BASE,POINT2[] " "}
DECL PDAT PP_OLP13={VEL 100.0,ACC 100.0,APO_DIST 100.0,APO_MODE #CDIS}
DECL E6POS Xp56={X 915.770081,Y 598.689575,Z 1493.11096,A 88.0728836,B 4.30365515,C -4.14981413,S 6,T 27,E1 0.0,E2 0.0,E3 0.0,E4 0.0,E5 0.0,E6 0.0}
DECL FDAT Fp57={TOOL_NO 2,BASE_NO 2,IPO_FRAME #BASE,POINT2[] " "}
DECL PDAT PP_OLP14={VEL 100.0,ACC 100.0,APO_DIST 100.0,APO_MODE #CDIS}
DECL E6POS Xp57={X 717.275879,Y 733.518127,Z 1267.56299,A 89.3907013,B 5.38819981,C -6.46229982,S 6,T 27,E1 0.0,E2 0.0,E3 0.0,E4 0.0,E5 0.0,E6 0.0}
DECL FDAT Fswp_60_1002={TOOL_NO 2,BASE_NO 2,IPO_FRAME #BASE,POINT2[] " "}
DECL PDAT PP_OLP15={VEL 60.0,ACC 100.0,APO_DIST 0.0}
DECL SPOT_TYPE SS_OLP4={GUN 2,PAIR #FIRST,RETR #CLO,CLO_TM 0,PGNO1 1,PRESS1 1.0,PGNO2 0,PRESS2 0.0}
DECL E6POS Xswp_60_1002={X 719.858521,Y 797.074219,Z 1273.64404,A 89.126442,B 5.25105381,C -6.19391298,S 6,T 27,E1 0.0,E2 0.0,E3 0.0,E4 0.0,E5 0.0,E6 0.0}
DECL FDAT Fp58={TOOL_NO 2,BASE_NO 2,IPO_FRAME #BASE,POINT2[] " "}
DECL PDAT PP_OLP16={VEL 100.0,ACC 100.0,APO_DIST 100.0,APO_MODE #CDIS}
DECL E6POS Xp58={X 717.145996,Y 733.567017,Z 1279.69299,A 89.3907013,B 5.38819981,C -6.46229982,S 6,T 27}
DECL FDAT Fp59={TOOL_NO 2,BASE_NO 2,IPO_FRAME #BASE,POINT2[] " "}
DECL PDAT PP_OLP17={VEL 100.0,ACC 100.0,APO_DIST 100.0,APO_MODE #CDIS}
DECL E6POS Xp59={X 973.581299,Y 724.721191,Z 1286.73303,A 91.3746567,B 0.503324926,C -4.664505,S 6,T 59,E1 0.0,E2 0.0,E3 0.0,E4 0.0,E5 0.0,E6 0.0}
DECL FDAT Fswp_60_1004={TOOL_NO 2,BASE_NO 2,IPO_FRAME #BASE,POINT2[] " "}
DECL SPOT_TYPE SS_OLP5={GUN 2,PAIR #FIRST,RETR #CLO,CLO_TM 0,PGNO1 1,PRESS1 1.0,PGNO2 0,PRESS2 0.0}
DECL E6POS Xswp_60_1004={X 971.583923,Y 800.74408,Z 1294.02295,A 109.672798,B 2.61476994,C -2.64917588,S 6,T 59,E1 0.0,E2 0.0,E3 0.0,E4 0.0,E5 0.0,E6 0.0}
DECL FDAT Fp61={TOOL_NO 2,BASE_NO 2,IPO_FRAME #BASE,POINT2[] " "}
DECL PDAT PP_OLP20={VEL 100.0,ACC 100.0,APO_DIST 100.0,APO_MODE #CDIS}
DECL E6POS Xp61={X 1048.60803,Y 694.463379,Z 1296.50403,A 110.633904,B 5.04574823,C -4.75294018,S 6,T 59,E1 0.0,E2 0.0,E3 0.0,E4 0.0,E5 0.0,E6 0.0}
DECL FDAT Fswp_60_1006={TOOL_NO 2,BASE_NO 2,IPO_FRAME #BASE,POINT2[] " "}
DECL PDAT PP_OLP21={VEL 60.0,ACC 100.0,APO_DIST 0.0}
DECL SPOT_TYPE SS_OLP6={GUN 2,PAIR #FIRST,RETR #CLO,CLO_TM 0,PGNO1 1,PRESS1 1.0,PGNO2 0,PRESS2 0.0}
DECL E6POS Xswp_60_1006={X 1252.11096,Y 805.172913,Z 1306.005,A 101.282204,B 1.45717597,C -2.17244792,S 6,T 57,E1 0.0,E2 0.0,E3 0.0,E4 0.0,E5 0.0,E6 0.0}
DECL FDAT Fp62={TOOL_NO 2,BASE_NO 2,IPO_FRAME #BASE,POINT2[] " "}
DECL PDAT PP_OLP22={VEL 100.0,ACC 100.0,APO_DIST 100.0,APO_MODE #CDIS}
DECL E6POS Xp62={X 1250.19495,Y 752.94397,Z 1303.40906,A 100.470596,B 4.95778179,C -1.97052002,S 6,T 57,E1 0.0,E2 0.0,E3 0.0,E4 0.0,E5 0.0,E6 0.0}
DECL FDAT Fp63={TOOL_NO 2,BASE_NO 2,IPO_FRAME #BASE,POINT2[] " "}
DECL PDAT PP_OLP23={VEL 100.0,ACC 100.0,APO_DIST 100.0,APO_MODE #CDIS}
DECL E6POS Xp63={X 993.91333,Y 706.072815,Z 1355.51697,A 100.4702,B 4.95808983,C -1.97126698,S 6,T 59,E1 0.0,E2 0.0,E3 0.0,E4 0.0,E5 0.0,E6 0.0}
DECL FDAT Fp64={TOOL_NO 2,BASE_NO 2,IPO_FRAME #BASE,POINT2[] " "}
DECL PDAT PP_OLP24={VEL 100.0,ACC 100.0,APO_DIST 100.0,APO_MODE #CDIS}
DECL E6POS Xp64={X 669.466309,Y 329.190796,Z 1536.40601,A 96.7606201,B 25.2837791,C 11.8137798,S 6,T 59,E1 0.0,E2 0.0,E3 0.0,E4 0.0,E5 0.0,E6 0.0}
DECL FDAT Fp65={TOOL_NO 2,BASE_NO 2,IPO_FRAME #BASE,POINT2[] " "}
DECL PDAT PP_OLP25={VEL 100.0,ACC 100.0,APO_DIST 0.0}
DECL E6POS Xp65={X 276.179413,Y 294.245392,Z 2159.01294,A 109.167198,B 21.4834003,C 42.7779198,S 6,T 59,E1 0.0,E2 0.0,E3 0.0,E4 0.0,E5 0.0,E6 0.0}
DECL SPOT_SUGG_T LAST_SPOT={GUN[] "1                       ",RETR_CMD[] "#OPN                    ",CHOISE[] "#FIRST                  ",CLO_TM[] "1                       ",PGNO1[] "1                       ",PRESS1[] "0                       ",PGNO2[] "1                       ",PRESS2[] "0                       ",SPOT_PARAMS[] "NORMAL                  "}
DECL E6POS XP1={X 812.945374,Y -138.445602,Z 1530.68506,A -140.2565,B 42.5539398,C -8.70740795,S 6,T 27,E1 0.0,E2 0.0,E3 0.0,E4 0.0,E5 0.0,E6 0.0}
DECL FDAT FP1={TOOL_NO 2,BASE_NO 2,IPO_FRAME #BASE,POINT2[] " ",TQ_STATE FALSE}
DECL PDAT PPDAT1={VEL 100.0,ACC 100.0,APO_DIST 100.0,APO_MODE #CDIS}
DECL LDAT LCPDAT1={VEL 1.0,ACC 100.0,APO_DIST 100.0,APO_FAC 50.0,AXIS_VEL 100.0,AXIS_ACC 100.0,ORI_TYP #VAR,CIRC_TYP #BASE,JERK_FAC 50.0,GEAR_JERK 50.0,EXAX_IGN 0}
DECL E6POS XP2={X 1070.36804,Y -728.833618,Z 1280.43201,A -74.2109528,B 0.4867872,C 2.79028702,S 2,T 10,E1 0.0,E2 0.0,E3 0.0,E4 0.0,E5 0.0,E6 0.0}
DECL FDAT FP2={TOOL_NO 2,BASE_NO 2,IPO_FRAME #BASE,POINT2[] " ",TQ_STATE FALSE}
DECL PDAT PPDAT2={VEL 100.0,ACC 100.0,APO_DIST 100.0,APO_MODE #CDIS}
DECL PDAT PPDAT3={VEL 100.0,ACC 100.0,APO_DIST 100.0,APO_MODE #CDIS}
DECL E6POS XP3={X 2868.28101,Y 2485.6521,Z 4716.08984,A 82.4006882,B -45.2431412,C -1.56597495,S 2,T 10,E1 0.0,E2 0.0,E3 0.0,E4 0.0,E5 0.0,E6 0.0}
DECL FDAT FP3={TOOL_NO 2,BASE_NO 1,IPO_FRAME #BASE,POINT2[] " ",TQ_STATE FALSE}
DECL PDAT PPDAT4={VEL 100.0,ACC 100.0,APO_DIST 100.0,APO_MODE #CDIS}
DECL E6POS XP4={X 814.124023,Y 41.7988205,Z 3106.80688,A -178.988297,B 40.6093292,C 0.315527499,S 2,T 2,E1 0.0,E2 0.0,E3 0.0,E4 0.0,E5 0.0,E6 0.0}
DECL FDAT FP4={TOOL_NO 2,BASE_NO 1,IPO_FRAME #BASE,POINT2[] " "}
DECL PDAT PPDAT5={VEL 100.0,ACC 100.0,APO_DIST 100.0,APO_MODE #CDIS}
DECL E6POS XP5={X 814.124023,Y 41.7988205,Z 3106.80688,A -178.988297,B 40.6093292,C 0.315527499,S 2,T 2,E1 0.0,E2 0.0,E3 0.0,E4 0.0,E5 0.0,E6 0.0}
DECL FDAT FP5={TOOL_NO 2,BASE_NO 1,IPO_FRAME #BASE,POINT2[] " "}
DECL PDAT PPDAT6={VEL 100.0,ACC 100.0,APO_DIST 100.0,APO_MODE #CDIS}
DECL E6POS XP6={X 2868.28101,Y 2485.6521,Z 4716.08984,A 82.4006882,B -45.2431412,C -1.56597495,S 2,T 10,E1 0.0,E2 0.0,E3 0.0,E4 0.0,E5 0.0,E6 0.0}
DECL FDAT FP6={TOOL_NO 2,BASE_NO 1,IPO_FRAME #BASE,POINT2[] " ",TQ_STATE FALSE}
DECL E6POS XP8={X 935.470886,Y -771.973877,Z 1405.79602,A -97.5937576,B 2.15295291,C 6.24414206,S 2,T 10,E1 0.0,E2 0.0,E3 0.0,E4 0.0,E5 0.0,E6 0.0}
DECL FDAT FP8={TOOL_NO 2,BASE_NO 1,IPO_FRAME #BASE,POINT2[] " ",TQ_STATE FALSE}
DECL PDAT PPDAT8={VEL 100.0,ACC 100.0,APO_DIST 100.0,APO_MODE #CDIS}
DECL E6POS XP10={X 1092.43201,Y 221.443207,Z 1495.92505,A 90.9198685,B -0.0189238694,C -4.79073811,S 6,T 59,E1 0.0,E2 0.0,E3 0.0,E4 0.0,E5 0.0,E6 0.0}
DECL FDAT FP10={TOOL_NO 2,BASE_NO 2,IPO_FRAME #BASE,POINT2[] " ",TQ_STATE FALSE}
DECL PDAT PPDAT10={VEL 100.0,ACC 100.0,APO_DIST 5.0,APO_MODE #CDIS}
DECL E6POS XP11={X 1093.37,Y 284.771393,Z 1324.06299,A 90.9199829,B -0.0188797805,C -4.79093504,S 6,T 59,E1 0.0,E2 0.0,E3 0.0,E4 0.0,E5 0.0,E6 0.0}
DECL FDAT FP11={TOOL_NO 2,BASE_NO 2,IPO_FRAME #BASE,POINT2[] " ",TQ_STATE FALSE}
DECL PDAT PPDAT11={VEL 100.0,ACC 100.0,APO_DIST 5.0,APO_MODE #CDIS}
DECL E6POS XP12={X 1092.56396,Y 349.022705,Z 1313.39197,A 90.9190674,B -0.0192148201,C -4.78931808,S 6,T 59,E1 0.0,E2 0.0,E3 0.0,E4 0.0,E5 0.0,E6 0.0}
DECL FDAT FP12={TOOL_NO 2,BASE_NO 2,IPO_FRAME #BASE,POINT2[] " ",TQ_STATE FALSE}
DECL PDAT PPDAT12={VEL 100.0,ACC 100.0,APO_DIST 5.0,APO_MODE #CDIS}
DECL E6POS XP13={X 1114.65503,Y 392.367615,Z 1304.48596,A 90.9190521,B -0.0194758102,C -4.78944778,S 6,T 59,E1 0.0,E2 0.0,E3 0.0,E4 0.0,E5 0.0,E6 0.0}
DECL FDAT FP13={TOOL_NO 2,BASE_NO 2,IPO_FRAME #BASE,POINT2[] " ",TQ_STATE FALSE}
DECL PDAT PPDAT13={VEL 100.0,ACC 100.0,APO_DIST 5.0,APO_MODE #CDIS}
DECL PDAT PPDAT14={VEL 60.0,ACC 100.0,APO_DIST 5.0,APO_MODE #CDIS}
DECL PDAT PPDAT15={VEL 60.0,ACC 100.0,APO_DIST 5.0,APO_MODE #CDIS}
DECL PDAT PPDAT16={VEL 60.0,ACC 100.0,APO_DIST 5.0,APO_MODE #CDIS}
DECL PDAT PPDAT17={VEL 60.0,ACC 100.0,APO_DIST 5.0,APO_MODE #CDIS}
DECL E6POS XP18={X 988.279724,Y 390.401489,Z 1289.36206,A 90.9188995,B -0.0173778906,C -4.78376198,S 6,T 59,E1 0.0,E2 0.0,E3 0.0,E4 0.0,E5 0.0,E6 0.0}
DECL FDAT FP18={TOOL_NO 2,BASE_NO 2,IPO_FRAME #BASE,POINT2[] " ",TQ_STATE FALSE}
DECL PDAT PPDAT18={VEL 100.0,ACC 100.0,APO_DIST 5.0,APO_MODE #CDIS}
DECL E6POS XP19={X 989.315002,Y 380.326508,Z 1297.75903,A 90.9190826,B 0.00535697909,C -4.78384686,S 6,T 59,E1 0.0,E2 0.0,E3 0.0,E4 0.0,E5 0.0,E6 0.0}
DECL FDAT FP19={TOOL_NO 2,BASE_NO 2,IPO_FRAME #BASE,POINT2[] " ",TQ_STATE FALSE}
DECL PDAT PPDAT19={VEL 100.0,ACC 100.0,APO_DIST 5.0,APO_MODE #CDIS}
DECL E6POS XP20={X 989.757202,Y 343.470703,Z 1307.48901,A 90.9157181,B 0.00516873784,C -4.78146076,S 6,T 59,E1 0.0,E2 0.0,E3 0.0,E4 0.0,E5 0.0,E6 0.0}
DECL FDAT FP20={TOOL_NO 2,BASE_NO 2,IPO_FRAME #BASE,POINT2[] " ",TQ_STATE FALSE}
DECL PDAT PPDAT20={VEL 100.0,ACC 100.0,APO_DIST 5.0,APO_MODE #CDIS}
DECL E6POS XP21={X 989.945618,Y 266.09491,Z 1394.34998,A 90.9181671,B 0.00415384397,C -4.78480005,S 6,T 27,E1 0.0,E2 0.0,E3 0.0,E4 0.0,E5 0.0,E6 0.0}
DECL FDAT FP21={TOOL_NO 2,BASE_NO 2,IPO_FRAME #BASE,POINT2[] " ",TQ_STATE FALSE}
DECL PDAT PPDAT21={VEL 100.0,ACC 100.0,APO_DIST 5.0,APO_MODE #CDIS}
DECL E6POS XP22={X 778.848328,Y 704.444275,Z 1587.37,A 113.120201,B 4.64594603,C -2.12198901,S 6,T 59,E1 0.0,E2 0.0,E3 0.0,E4 0.0,E5 0.0,E6 0.0}
DECL FDAT FP22={TOOL_NO 2,BASE_NO 2,IPO_FRAME #BASE,POINT2[] " ",TQ_STATE FALSE}
DECL PDAT PPDAT22={VEL 100.0,ACC 100.0,APO_DIST 5.0,APO_MODE #CDIS}
DECL E6POS XP23={X 644.905212,Y 225.569595,Z 1724.90906,A -173.402603,B 32.6836319,C 1.02964699,S 6,T 50,E1 0.0,E2 0.0,E3 0.0,E4 0.0,E5 0.0,E6 0.0}
DECL FDAT FP23={TOOL_NO 2,BASE_NO 2,IPO_FRAME #BASE,POINT2[] " ",TQ_STATE FALSE}
DECL PDAT PPDAT23={VEL 100.0,ACC 100.0,APO_DIST 5.0,APO_MODE #CDIS}
DECL E6POS XP24={X 935.841309,Y -123.237396,Z 1682.49194,A -89.9244232,B 0.906739712,C 2.82238603,S 6,T 18,E1 0.0,E2 0.0,E3 0.0,E4 0.0,E5 0.0,E6 0.0}
DECL FDAT FP24={TOOL_NO 2,BASE_NO 2,IPO_FRAME #BASE,POINT2[] " ",TQ_STATE FALSE}
DECL PDAT PPDAT24={VEL 100.0,ACC 100.0,APO_DIST 5.0,APO_MODE #CDIS}
DECL E6POS XP25={X 1101.95398,Y 578.030212,Z 1409.16699,A -73.3142166,B 2.35896611,C 4.18486309,S 6,T 18,E1 0.0,E2 0.0,E3 0.0,E4 0.0,E5 0.0,E6 0.0}
DECL FDAT FP25={TOOL_NO 2,BASE_NO 2,IPO_FRAME #BASE,POINT2[] " ",TQ_STATE FALSE}
DECL PDAT PPDAT25={VEL 100.0,ACC 100.0,APO_DIST 5.0,APO_MODE #CDIS}
DECL E6POS XP26={X 1103.21594,Y 557.477783,Z 1317.85303,A -73.3879929,B 1.87317801,C 5.91192198,S 6,T 18,E1 0.0,E2 0.0,E3 0.0,E4 0.0,E5 0.0,E6 0.0}
DECL FDAT FP26={TOOL_NO 2,BASE_NO 2,IPO_FRAME #BASE,POINT2[] " ",TQ_STATE FALSE}
DECL PDAT PPDAT26={VEL 100.0,ACC 100.0,APO_DIST 5.0,APO_MODE #CDIS}
DECL E6POS XP27={X 1103.85498,Y 514.706909,Z 1314.76501,A -73.387558,B 1.87311399,C 5.91158915,S 6,T 18,E1 0.0,E2 0.0,E3 0.0,E4 0.0,E5 0.0,E6 0.0}
DECL FDAT FP27={TOOL_NO 2,BASE_NO 2,IPO_FRAME #BASE,POINT2[] " ",TQ_STATE FALSE}
DECL PDAT PPDAT27={VEL 100.0,ACC 100.0,APO_DIST 5.0,APO_MODE #CDIS}
DECL E6POS XP28={X 1104.16504,Y 496.300293,Z 1309.63306,A -73.3874969,B 1.87330198,C 5.91125393,S 6,T 18,E1 0.0,E2 0.0,E3 0.0,E4 0.0,E5 0.0,E6 0.0}
DECL FDAT FP28={TOOL_NO 2,BASE_NO 2,IPO_FRAME #BASE,POINT2[] " ",TQ_STATE FALSE}
DECL PDAT PPDAT28={VEL 100.0,ACC 100.0,APO_DIST 5.0,APO_MODE #CDIS}
DECL E6POS XP29={X 1104.71997,Y 470.117798,Z 1292.14001,A -73.3867798,B 1.87337196,C 5.910501,S 6,T 18,E1 0.0,E2 0.0,E3 0.0,E4 0.0,E5 0.0,E6 0.0}
DECL FDAT FP29={TOOL_NO 2,BASE_NO 2,IPO_FRAME #BASE,POINT2[] " ",TQ_STATE FALSE}
DECL PDAT PPDAT29={VEL 100.0,ACC 100.0,APO_DIST 5.0,APO_MODE #CDIS}
DECL E6POS XP30={X 1168.17505,Y 454.355591,Z 1298.62195,A -73.7040863,B -2.84922409,C 4.26323986,S 6,T 18,E1 0.0,E2 0.0,E3 0.0,E4 0.0,E5 0.0,E6 0.0}
DECL FDAT FP30={TOOL_NO 2,BASE_NO 2,IPO_FRAME #BASE,POINT2[] " ",TQ_STATE FALSE}
DECL PDAT PPDAT30={VEL 100.0,ACC 100.0,APO_DIST 5.0,APO_MODE #CDIS}
DECL PDAT PPDAT31={VEL 60.0,ACC 100.0,APO_DIST 5.0,APO_MODE #CDIS}
DECL E6POS XP32={X 1147.06995,Y 454.036804,Z 1301.09998,A -73.6426163,B -3.62066698,C 1.499421,S 6,T 18,E1 0.0,E2 0.0,E3 0.0,E4 0.0,E5 0.0,E6 0.0}
DECL FDAT FP32={TOOL_NO 2,BASE_NO 2,IPO_FRAME #BASE,POINT2[] " ",TQ_STATE FALSE}
DECL PDAT PPDAT32={VEL 100.0,ACC 100.0,APO_DIST 5.0,APO_MODE #CDIS}
DECL PDAT PPDAT33={VEL 60.0,ACC 100.0,APO_DIST 5.0,APO_MODE #CDIS}
DECL E6POS XP34={X 1103.16699,Y 453.236389,Z 1300.63599,A -74.2926788,B -4.11864185,C 1.33635604,S 6,T 18,E1 0.0,E2 0.0,E3 0.0,E4 0.0,E5 0.0,E6 0.0}
DECL FDAT FP34={TOOL_NO 2,BASE_NO 2,IPO_FRAME #BASE,POINT2[] " ",TQ_STATE FALSE}
DECL PDAT PPDAT34={VEL 100.0,ACC 100.0,APO_DIST 5.0,APO_MODE #CDIS}
DECL PDAT PPDAT35={VEL 60.0,ACC 100.0,APO_DIST 5.0,APO_MODE #CDIS}
DECL E6POS XP36={X 1057.23096,Y 452.561798,Z 1293.505,A -74.3145065,B -2.03506804,C 2.11838698,S 6,T 18,E1 0.0,E2 0.0,E3 0.0,E4 0.0,E5 0.0,E6 0.0}
DECL FDAT FP36={TOOL_NO 2,BASE_NO 2,IPO_FRAME #BASE,POINT2[] " ",TQ_STATE FALSE}
DECL PDAT PPDAT36={VEL 100.0,ACC 100.0,APO_DIST 5.0,APO_MODE #CDIS}
DECL PDAT PPDAT37={VEL 60.0,ACC 100.0,APO_DIST 5.0,APO_MODE #CDIS}
DECL E6POS XP38={X 1036.104,Y 464.092987,Z 1288.23901,A -73.9398117,B -1.62330496,C 5.2520771,S 6,T 18,E1 0.0,E2 0.0,E3 0.0,E4 0.0,E5 0.0,E6 0.0}
DECL FDAT FP38={TOOL_NO 2,BASE_NO 2,IPO_FRAME #BASE,POINT2[] " ",TQ_STATE FALSE}
DECL PDAT PPDAT38={VEL 100.0,ACC 100.0,APO_DIST 5.0,APO_MODE #CDIS}
DECL E6POS XP39={X 1035.51001,Y 492.406097,Z 1305.92505,A -73.940239,B -1.62303805,C 5.25236416,S 6,T 18,E1 0.0,E2 0.0,E3 0.0,E4 0.0,E5 0.0,E6 0.0}
DECL FDAT FP39={TOOL_NO 2,BASE_NO 2,IPO_FRAME #BASE,POINT2[] " ",TQ_STATE FALSE}
DECL PDAT PPDAT39={VEL 100.0,ACC 100.0,APO_DIST 5.0,APO_MODE #CDIS}
DECL E6POS XP40={X 1035.10095,Y 516.023499,Z 1313.36304,A -73.8458862,B 4.08358002,C 6.80825615,S 6,T 50,E1 0.0,E2 0.0,E3 0.0,E4 0.0,E5 0.0,E6 0.0}
DECL FDAT FP40={TOOL_NO 2,BASE_NO 2,IPO_FRAME #BASE,POINT2[] " ",TQ_STATE FALSE}
DECL PDAT PPDAT40={VEL 100.0,ACC 100.0,APO_DIST 5.0,APO_MODE #CDIS}
DECL E6POS XP41={X 1034.73206,Y 538.545288,Z 1316.14502,A -73.7335434,B 7.12919617,C 7.64717197,S 6,T 50,E1 0.0,E2 0.0,E3 0.0,E4 0.0,E5 0.0,E6 0.0}
DECL FDAT FP41={TOOL_NO 2,BASE_NO 2,IPO_FRAME #BASE,POINT2[] " ",TQ_STATE FALSE}
DECL PDAT PPDAT41={VEL 100.0,ACC 100.0,APO_DIST 5.0,APO_MODE #CDIS}
DECL E6POS XP42={X 1033.177,Y 578.153992,Z 1414.33997,A -73.2801132,B 14.1782799,C 9.67325592,S 6,T 50,E1 0.0,E2 0.0,E3 0.0,E4 0.0,E5 0.0,E6 0.0}
DECL FDAT FP42={TOOL_NO 2,BASE_NO 2,IPO_FRAME #BASE,POINT2[] " ",TQ_STATE FALSE}
DECL PDAT PPDAT42={VEL 100.0,ACC 100.0,APO_DIST 5.0,APO_MODE #CDIS}
DECL E6POS XP43={X 928.931274,Y -76.4975128,Z 1822.14795,A -110.113899,B 3.72326708,C 7.68550682,S 6,T 18,E1 0.0,E2 0.0,E3 0.0,E4 0.0,E5 0.0,E6 0.0}
DECL FDAT FP43={TOOL_NO 2,BASE_NO 2,IPO_FRAME #BASE,POINT2[] " ",TQ_STATE FALSE}
DECL PDAT PPDAT43={VEL 100.0,ACC 100.0,APO_DIST 5.0,APO_MODE #CDIS}
DECL E6POS XP44={X 981.711914,Y 337.245911,Z 1469.375,A 113.450996,B 47.8786888,C -2.15183306,S 6,T 50,E1 0.0,E2 0.0,E3 0.0,E4 0.0,E5 0.0,E6 0.0}
DECL FDAT FP44={TOOL_NO 2,BASE_NO 2,IPO_FRAME #BASE,POINT2[] " ",TQ_STATE FALSE}
DECL PDAT PPDAT44={VEL 100.0,ACC 100.0,APO_DIST 5.0,APO_MODE #CDIS}
DECL E6POS XP45={X 1097.39294,Y 393.750397,Z 1296.12598,A 90.8787231,B 3.72913504,C -4.77820206,S 6,T 59,E1 0.0,E2 0.0,E3 0.0,E4 0.0,E5 0.0,E6 0.0}
DECL FDAT FP45={TOOL_NO 2,BASE_NO 2,IPO_FRAME #BASE,POINT2[] " ",TQ_STATE FALSE}
DECL PDAT PPDAT45={VEL 100.0,ACC 100.0,APO_DIST 5.0,APO_MODE #CDIS}
DECL E6POS XP46={X 1055.56396,Y 391.366608,Z 1294.68103,A 90.8883896,B 2.73829007,C -4.77724409,S 6,T 59,E1 0.0,E2 0.0,E3 0.0,E4 0.0,E5 0.0,E6 0.0}
DECL FDAT FP46={TOOL_NO 2,BASE_NO 2,IPO_FRAME #BASE,POINT2[] " ",TQ_STATE FALSE}
DECL PDAT PPDAT46={VEL 100.0,ACC 100.0,APO_DIST 5.0,APO_MODE #CDIS}
DECL E6POS XP66={X 1010.84399,Y 390.599091,Z 1294.04602,A 90.8889008,B 2.85570097,C -4.78140116,S 6,T 59,E1 0.0,E2 0.0,E3 0.0,E4 0.0,E5 0.0,E6 0.0}
DECL FDAT FP66={TOOL_NO 2,BASE_NO 2,IPO_FRAME #BASE,POINT2[] " ",TQ_STATE FALSE}
DECL PDAT PPDAT47={VEL 100.0,ACC 100.0,APO_DIST 5.0,APO_MODE #CDIS}
DECL E6POS XP67={X 1105.24097,Y 265.770508,Z 1547.04102,A 162.211899,B 56.1322403,C 3.32080698,S 2,T 10,E1 0.0,E2 0.0,E3 0.0,E4 0.0,E5 0.0,E6 0.0}
DECL FDAT FP67={TOOL_NO 2,BASE_NO 2,IPO_FRAME #BASE,POINT2[] " ",TQ_STATE FALSE}
DECL PDAT PPDAT48={VEL 100.0,ACC 100.0,APO_DIST 5.0,APO_MODE #CDIS}
DECL E6POS XSwp_65_0004={X 1125.16394,Y 394.060303,Z 1310.99805,A 91.163208,B 4.51505518,C -3.36029601,S 6,T 59,E1 0.0,E2 0.0,E3 0.0,E4 0.0,E5 0.0,E6 0.0}
DECL FDAT FSwp_65_0004={TOOL_NO 2,BASE_NO 2,IPO_FRAME #BASE,POINT2[] " ",TQ_STATE FALSE}
DECL E6POS XSwp_65_0006={X 1077.53198,Y 393.541687,Z 1308.50598,A 91.0277786,B 3.72262406,C -2.34453011,S 6,T 59,E1 0.0,E2 0.0,E3 0.0,E4 0.0,E5 0.0,E6 0.0}
DECL FDAT FSwp_65_0006={TOOL_NO 2,BASE_NO 2,IPO_FRAME #BASE,POINT2[] " ",TQ_STATE FALSE}
DECL E6POS XSwp_65_0008={X 1031.56897,Y 391.072113,Z 1305.69897,A 90.9567337,B 2.73596001,C -3.19474602,S 6,T 59,E1 0.0,E2 0.0,E3 0.0,E4 0.0,E5 0.0,E6 0.0}
DECL FDAT FSwp_65_0008={TOOL_NO 2,BASE_NO 2,IPO_FRAME #BASE,POINT2[] " ",TQ_STATE FALSE}
DECL E6POS XSwp_65_0010={X 987.183411,Y 391.4599,Z 1303.55603,A 90.9280167,B 2.85265899,C -3.93145895,S 6,T 59,E1 0.0,E2 0.0,E3 0.0,E4 0.0,E5 0.0,E6 0.0}
DECL FDAT FSwp_65_0010={TOOL_NO 2,BASE_NO 2,IPO_FRAME #BASE,POINT2[] " ",TQ_STATE FALSE}
DECL E6POS XSwp_65_0001={X 1168.10498,Y 454.370514,Z 1309.63098,A -73.6425171,B -3.62056494,C 1.49930501,S 6,T 18,E1 0.0,E2 0.0,E3 0.0,E4 0.0,E5 0.0,E6 0.0}
DECL FDAT FSwp_65_0001={TOOL_NO 2,BASE_NO 2,IPO_FRAME #BASE,POINT2[] " ",TQ_STATE FALSE}
DECL E6POS XSwp_65_0003={X 1129.46399,Y 453.495392,Z 1308.10303,A -74.2948227,B -3.85864592,C 1.40684295,S 6,T 18,E1 0.0,E2 0.0,E3 0.0,E4 0.0,E5 0.0,E6 0.0}
DECL FDAT FSwp_65_0003={TOOL_NO 2,BASE_NO 2,IPO_FRAME #BASE,POINT2[] " ",TQ_STATE FALSE}
DECL E6POS XSwp_65_0005={X 1080.36499,Y 452.933289,Z 1305.97705,A -74.3143997,B -2.03536701,C 2.11848998,S 6,T 18,E1 0.0,E2 0.0,E3 0.0,E4 0.0,E5 0.0,E6 0.0}
DECL FDAT FSwp_65_0005={TOOL_NO 2,BASE_NO 2,IPO_FRAME #BASE,POINT2[] " ",TQ_STATE FALSE}
DECL E6POS XSwp_65_0007={X 1037.50903,Y 452.317993,Z 1303.33301,A -74.3151169,B -2.03562808,C 2.11908698,S 6,T 18,E1 0.0,E2 0.0,E3 0.0,E4 0.0,E5 0.0,E6 0.0}
DECL FDAT FSwp_65_0007={TOOL_NO 2,BASE_NO 2,IPO_FRAME #BASE,POINT2[] " ",TQ_STATE FALSE}
DECL PDAT PPDAT0={VEL 100.0,ACC 100.0,APO_DIST 100.0,APO_MODE #CDIS}
DECL E6POS XP0={X 1022.73499,Y -738.125427,Z 2042.82397,A -70.2032394,B 12.54422,C 18.9223194,S 2,T 11,E1 0.0,E2 0.0,E3 0.0,E4 0.0,E5 0.0,E6 0.0}
DECL FDAT FP0={TOOL_NO 2,BASE_NO 1,IPO_FRAME #BASE,POINT2[] " "}
ENDDAT
